  PROC DrawPart288()
    MoveL Offs(pOrigin,140.46,85.96,6.00),v60,z5,tPen\WObj:=wPaper;
    MoveL Offs(pOrigin,136.24,84.26,6.00),vTravel,z5,tPen\WObj:=wPaper;
    MoveL Offs(pOrigin,136.24,84.26,0.00),v60,z0,tPen\WObj:=wPaper;
    MoveL Offs(pOrigin,134.58,82.61,0.00),v40,z0,tPen\WObj:=wPaper;
    MoveL Offs(pOrigin,134.40,83.64,0.00),v40,z0,tPen\WObj:=wPaper;
    MoveL Offs(pOrigin,127.18,83.64,0.00),v40,z0,tPen\WObj:=wPaper;
    MoveL Offs(pOrigin,127.70,84.68,0.00),v40,z0,tPen\WObj:=wPaper;
    MoveL Offs(pOrigin,123.49,80.48,0.00),v40,fine,tPen\WObj:=wPaper;
    MoveL Offs(pOrigin,123.49,80.48,6.00),v60,z5,tPen\WObj:=wPaper;
    MoveL Offs(pOrigin,124.41,82.58,6.00),vTravel,z5,tPen\WObj:=wPaper;
    MoveL Offs(pOrigin,124.41,82.58,0.00),v60,z0,tPen\WObj:=wPaper;
    MoveL Offs(pOrigin,130.57,82.58,0.00),v40,z0,tPen\WObj:=wPaper;
    MoveL Offs(pOrigin,130.51,81.80,0.00),v40,z0,tPen\WObj:=wPaper;
    MoveL Offs(pOrigin,127.35,84.96,0.00),v40,fine,tPen\WObj:=wPaper;
    MoveL Offs(pOrigin,127.35,84.96,6.00),v60,z5,tPen\WObj:=wPaper;
    MoveL Offs(pOrigin,125.90,82.35,6.00),vTravel,z5,tPen\WObj:=wPaper;
    MoveL Offs(pOrigin,125.90,82.35,0.00),v60,z0,tPen\WObj:=wPaper;
    MoveL Offs(pOrigin,125.69,81.85,0.00),v40,z0,tPen\WObj:=wPaper;
    MoveL Offs(pOrigin,122.07,80.08,0.00),v40,z0,tPen\WObj:=wPaper;
    MoveL Offs(pOrigin,118.25,77.68,0.00),v40,z0,tPen\WObj:=wPaper;
    MoveL Offs(pOrigin,112.72,73.00,0.00),v40,fine,tPen\WObj:=wPaper;
    MoveL Offs(pOrigin,112.72,73.00,6.00),v60,z5,tPen\WObj:=wPaper;
    MoveL Offs(pOrigin,108.90,73.00,6.00),vTravel,z5,tPen\WObj:=wPaper;
    MoveL Offs(pOrigin,108.90,73.00,0.00),v60,z0,tPen\WObj:=wPaper;
    MoveL Offs(pOrigin,109.11,73.43,0.00),v40,z0,tPen\WObj:=wPaper;
    MoveL Offs(pOrigin,108.90,73.00,0.00),v40,fine,tPen\WObj:=wPaper;
    MoveL Offs(pOrigin,108.90,73.00,6.00),v60,z5,tPen\WObj:=wPaper;
    MoveL Offs(pOrigin,106.27,71.69,6.00),vTravel,z5,tPen\WObj:=wPaper;
    MoveL Offs(pOrigin,106.27,71.69,0.00),v60,z0,tPen\WObj:=wPaper;
    MoveL Offs(pOrigin,107.62,70.34,0.00),v40,z0,tPen\WObj:=wPaper;
    MoveL Offs(pOrigin,106.88,69.59,0.00),v40,z0,tPen\WObj:=wPaper;
    MoveL Offs(pOrigin,105.68,70.80,0.00),v40,z0,tPen\WObj:=wPaper;
    MoveL Offs(pOrigin,104.93,70.05,0.00),v40,z0,tPen\WObj:=wPaper;
    MoveL Offs(pOrigin,106.13,68.85,0.00),v40,z0,tPen\WObj:=wPaper;
    MoveL Offs(pOrigin,105.53,67.95,0.00),v40,z0,tPen\WObj:=wPaper;
    MoveL Offs(pOrigin,104.18,69.30,0.00),v40,fine,tPen\WObj:=wPaper;
    MoveL Offs(pOrigin,104.18,69.30,6.00),v60,z5,tPen\WObj:=wPaper;
    MoveL Offs(pOrigin,104.64,67.35,6.00),vTravel,z5,tPen\WObj:=wPaper;
    MoveL Offs(pOrigin,104.64,67.35,0.00),v60,z0,tPen\WObj:=wPaper;
    MoveL Offs(pOrigin,101.18,70.81,0.00),v40,z0,tPen\WObj:=wPaper;
    MoveL Offs(pOrigin,101.29,70.22,0.00),v40,z0,tPen\WObj:=wPaper;
    MoveL Offs(pOrigin,103.69,72.63,0.00),v40,fine,tPen\WObj:=wPaper;
    MoveL Offs(pOrigin,103.69,72.63,6.00),v60,z5,tPen\WObj:=wPaper;
    MoveL Offs(pOrigin,104.77,73.20,6.00),vTravel,z5,tPen\WObj:=wPaper;
    MoveL Offs(pOrigin,104.77,73.20,0.00),v60,z0,tPen\WObj:=wPaper;
    MoveL Offs(pOrigin,103.27,74.70,0.00),v40,z0,tPen\WObj:=wPaper;
    MoveL Offs(pOrigin,103.86,75.59,0.00),v40,z0,tPen\WObj:=wPaper;
    MoveL Offs(pOrigin,105.37,74.09,0.00),v40,z0,tPen\WObj:=wPaper;
    MoveL Offs(pOrigin,105.96,74.99,0.00),v40,z0,tPen\WObj:=wPaper;
    MoveL Offs(pOrigin,104.46,76.49,0.00),v40,fine,tPen\WObj:=wPaper;
    MoveL Offs(pOrigin,104.46,76.49,6.00),v60,z5,tPen\WObj:=wPaper;
    MoveL Offs(pOrigin,101.04,77.89,6.00),vTravel,z5,tPen\WObj:=wPaper;
    MoveL Offs(pOrigin,101.04,77.89,0.00),v60,z0,tPen\WObj:=wPaper;
    MoveL Offs(pOrigin,100.61,76.61,0.00),v40,z0,tPen\WObj:=wPaper;
    MoveL Offs(pOrigin,95.51,71.16,0.00),v40,z0,tPen\WObj:=wPaper;
    MoveL Offs(pOrigin,94.52,70.66,0.00),v40,z0,tPen\WObj:=wPaper;
    MoveL Offs(pOrigin,92.89,67.69,0.00),v40,z0,tPen\WObj:=wPaper;
    MoveL Offs(pOrigin,92.54,66.41,0.00),v40,z0,tPen\WObj:=wPaper;
    MoveL Offs(pOrigin,92.21,66.34,0.00),v40,z0,tPen\WObj:=wPaper;
    MoveL Offs(pOrigin,88.45,70.10,0.00),v40,fine,tPen\WObj:=wPaper;
    MoveL Offs(pOrigin,88.45,70.10,6.00),v60,z5,tPen\WObj:=wPaper;
    MoveL Offs(pOrigin,88.60,71.45,6.00),vTravel,z5,tPen\WObj:=wPaper;
    MoveL Offs(pOrigin,88.60,71.45,0.00),v60,z0,tPen\WObj:=wPaper;
    MoveL Offs(pOrigin,93.25,66.79,0.00),v40,fine,tPen\WObj:=wPaper;
    MoveL Offs(pOrigin,93.25,66.79,6.00),v60,z5,tPen\WObj:=wPaper;
    MoveL Offs(pOrigin,91.76,65.30,6.00),vTravel,z5,tPen\WObj:=wPaper;
    MoveL Offs(pOrigin,91.76,65.30,0.00),v60,z0,tPen\WObj:=wPaper;
    MoveL Offs(pOrigin,88.46,68.60,0.00),v40,z0,tPen\WObj:=wPaper;
    MoveL Offs(pOrigin,89.35,68.86,0.00),v40,z0,tPen\WObj:=wPaper;
    MoveL Offs(pOrigin,90.84,68.86,0.00),v40,fine,tPen\WObj:=wPaper;
    MoveL Offs(pOrigin,90.84,68.86,6.00),v60,z5,tPen\WObj:=wPaper;
    MoveL Offs(pOrigin,88.31,67.25,6.00),vTravel,z5,tPen\WObj:=wPaper;
    MoveL Offs(pOrigin,88.31,67.25,0.00),v60,z0,tPen\WObj:=wPaper;
    MoveL Offs(pOrigin,91.92,63.65,0.00),v40,fine,tPen\WObj:=wPaper;
    MoveL Offs(pOrigin,91.92,63.65,6.00),v60,z5,tPen\WObj:=wPaper;
    MoveL Offs(pOrigin,92.37,61.70,6.00),vTravel,z5,tPen\WObj:=wPaper;
    MoveL Offs(pOrigin,92.37,61.70,0.00),v60,z0,tPen\WObj:=wPaper;
    MoveL Offs(pOrigin,88.46,65.61,0.00),v40,z0,tPen\WObj:=wPaper;
    MoveL Offs(pOrigin,89.35,65.69,0.00),v40,z0,tPen\WObj:=wPaper;
    MoveL Offs(pOrigin,90.84,65.69,0.00),v40,fine,tPen\WObj:=wPaper;
    MoveL Offs(pOrigin,90.84,65.69,6.00),v60,z5,tPen\WObj:=wPaper;
    MoveL Offs(pOrigin,94.77,62.29,6.00),vTravel,z5,tPen\WObj:=wPaper;
    MoveL Offs(pOrigin,94.77,62.29,0.00),v60,z0,tPen\WObj:=wPaper;
    MoveL Offs(pOrigin,98.22,58.83,0.00),v40,z0,tPen\WObj:=wPaper;
    MoveL Offs(pOrigin,97.36,58.82,0.00),v40,z0,tPen\WObj:=wPaper;
    MoveL Offs(pOrigin,91.80,53.26,0.00),v40,z0,tPen\WObj:=wPaper;
    MoveL Offs(pOrigin,92.32,53.02,0.00),v40,z0,tPen\WObj:=wPaper;
    MoveL Offs(pOrigin,94.66,53.02,0.00),v40,z0,tPen\WObj:=wPaper;
    MoveL Offs(pOrigin,95.55,52.55,0.00),v40,z0,tPen\WObj:=wPaper;
    MoveL Offs(pOrigin,89.54,58.56,0.00),v40,fine,tPen\WObj:=wPaper;
    MoveL Offs(pOrigin,89.54,58.56,6.00),v60,z5,tPen\WObj:=wPaper;
    MoveL Offs(pOrigin,91.05,57.24,6.00),vTravel,z5,tPen\WObj:=wPaper;
    MoveL Offs(pOrigin,91.05,57.24,0.00),v60,z0,tPen\WObj:=wPaper;
    MoveL Offs(pOrigin,95.30,57.24,0.00),v40,z0,tPen\WObj:=wPaper;
    MoveL Offs(pOrigin,95.30,56.18,0.00),v40,z0,tPen\WObj:=wPaper;
    MoveL Offs(pOrigin,91.48,56.18,0.00),v40,z0,tPen\WObj:=wPaper;
    MoveL Offs(pOrigin,91.06,55.51,0.00),v40,z0,tPen\WObj:=wPaper;
    MoveL Offs(pOrigin,101.13,65.58,0.00),v40,z0,tPen\WObj:=wPaper;
    MoveL Offs(pOrigin,102.10,65.41,0.00),v40,z0,tPen\WObj:=wPaper;
    MoveL Offs(pOrigin,99.54,67.97,0.00),v40,z0,tPen\WObj:=wPaper;
    MoveL Offs(pOrigin,100.14,68.87,0.00),v40,z0,tPen\WObj:=wPaper;
    MoveL Offs(pOrigin,102.84,66.16,0.00),v40,z0,tPen\WObj:=wPaper;
    MoveL Offs(pOrigin,103.74,66.76,0.00),v40,z0,tPen\WObj:=wPaper;
    MoveL Offs(pOrigin,100.74,69.76,0.00),v40,fine,tPen\WObj:=wPaper;
    MoveL Offs(pOrigin,100.74,69.76,6.00),v60,z5,tPen\WObj:=wPaper;
    MoveL Offs(pOrigin,101.58,67.53,6.00),vTravel,z5,tPen\WObj:=wPaper;
    MoveL Offs(pOrigin,101.58,67.53,0.00),v60,z0,tPen\WObj:=wPaper;
    MoveL Offs(pOrigin,90.76,56.71,0.00),v40,z0,tPen\WObj:=wPaper;
    MoveL Offs(pOrigin,90.29,56.31,0.00),v40,z0,tPen\WObj:=wPaper;
    MoveL Offs(pOrigin,95.25,51.35,0.00),v40,fine,tPen\WObj:=wPaper;
    MoveL Offs(pOrigin,95.25,51.35,6.00),v60,z5,tPen\WObj:=wPaper;
    MoveL Offs(pOrigin,94.24,49.85,6.00),vTravel,z5,tPen\WObj:=wPaper;
    MoveL Offs(pOrigin,94.24,49.85,0.00),v60,z0,tPen\WObj:=wPaper;
    MoveL Offs(pOrigin,92.32,49.85,0.00),v40,fine,tPen\WObj:=wPaper;
    MoveL Offs(pOrigin,92.32,49.85,6.00),v60,z5,tPen\WObj:=wPaper;
    MoveL Offs(pOrigin,91.36,50.77,6.00),vTravel,z5,tPen\WObj:=wPaper;
    MoveL Offs(pOrigin,91.36,50.77,0.00),v60,z0,tPen\WObj:=wPaper;
    MoveL Offs(pOrigin,95.56,46.56,0.00),v40,z0,tPen\WObj:=wPaper;
    MoveL Offs(pOrigin,94.45,46.68,0.00),v40,z0,tPen\WObj:=wPaper;
    MoveL Offs(pOrigin,93.18,46.68,0.00),v40,fine,tPen\WObj:=wPaper;
  ENDPROC

  PROC DrawPart289()
    MoveL Offs(pOrigin,93.18,46.68,6.00),v60,z5,tPen\WObj:=wPaper;
    MoveL Offs(pOrigin,94.24,44.57,6.00),vTravel,z5,tPen\WObj:=wPaper;
    MoveL Offs(pOrigin,94.24,44.57,0.00),v60,z0,tPen\WObj:=wPaper;
    MoveL Offs(pOrigin,95.94,44.57,0.00),v40,z0,tPen\WObj:=wPaper;
    MoveL Offs(pOrigin,96.57,44.59,0.00),v40,z0,tPen\WObj:=wPaper;
    MoveL Offs(pOrigin,95.22,43.24,0.00),v40,z0,tPen\WObj:=wPaper;
    MoveL Offs(pOrigin,95.30,43.51,0.00),v40,z0,tPen\WObj:=wPaper;
    MoveL Offs(pOrigin,97.00,43.51,0.00),v40,z0,tPen\WObj:=wPaper;
    MoveL Offs(pOrigin,97.00,43.67,0.00),v40,z0,tPen\WObj:=wPaper;
    MoveL Offs(pOrigin,95.51,45.16,0.00),v40,z0,tPen\WObj:=wPaper;
    MoveL Offs(pOrigin,97.00,43.67,0.00),v40,z0,tPen\WObj:=wPaper;
    MoveL Offs(pOrigin,97.46,43.99,0.00),v40,z0,tPen\WObj:=wPaper;
    MoveL Offs(pOrigin,95.81,42.34,0.00),v40,z0,tPen\WObj:=wPaper;
    MoveL Offs(pOrigin,95.94,42.61,0.00),v40,z0,tPen\WObj:=wPaper;
    MoveL Offs(pOrigin,94.03,44.53,0.00),v40,z0,tPen\WObj:=wPaper;
    MoveL Offs(pOrigin,95.94,42.61,0.00),v40,fine,tPen\WObj:=wPaper;
    MoveL Offs(pOrigin,95.94,42.61,6.00),v60,z5,tPen\WObj:=wPaper;
    MoveL Offs(pOrigin,97.64,41.55,6.00),vTravel,z5,tPen\WObj:=wPaper;
    MoveL Offs(pOrigin,97.64,41.55,0.00),v60,z0,tPen\WObj:=wPaper;
    MoveL Offs(pOrigin,99.55,40.42,0.00),v40,z0,tPen\WObj:=wPaper;
    MoveL Offs(pOrigin,106.35,38.58,0.00),v40,z0,tPen\WObj:=wPaper;
    MoveL Offs(pOrigin,106.67,39.00,0.00),v40,z0,tPen\WObj:=wPaper;
    MoveL Offs(pOrigin,106.67,40.06,0.00),v40,fine,tPen\WObj:=wPaper;
    MoveL Offs(pOrigin,106.67,40.06,6.00),v60,z5,tPen\WObj:=wPaper;
    MoveL Offs(pOrigin,108.78,40.49,6.00),vTravel,z5,tPen\WObj:=wPaper;
    MoveL Offs(pOrigin,108.78,40.49,0.00),v60,z0,tPen\WObj:=wPaper;
    MoveL Offs(pOrigin,108.78,37.72,0.00),v40,z0,tPen\WObj:=wPaper;
    MoveL Offs(pOrigin,109.84,37.72,0.00),v40,z0,tPen\WObj:=wPaper;
    MoveL Offs(pOrigin,109.84,39.85,0.00),v40,fine,tPen\WObj:=wPaper;
    MoveL Offs(pOrigin,109.84,39.85,6.00),v60,z5,tPen\WObj:=wPaper;
    MoveL Offs(pOrigin,109.44,41.04,6.00),vTravel,z5,tPen\WObj:=wPaper;
    MoveL Offs(pOrigin,109.44,41.04,0.00),v60,z0,tPen\WObj:=wPaper;
    MoveL Offs(pOrigin,104.48,36.08,0.00),v40,fine,tPen\WObj:=wPaper;
    MoveL Offs(pOrigin,104.48,36.08,6.00),v60,z5,tPen\WObj:=wPaper;
    MoveL Offs(pOrigin,103.69,33.95,6.00),vTravel,z5,tPen\WObj:=wPaper;
    MoveL Offs(pOrigin,103.69,33.95,0.00),v60,z0,tPen\WObj:=wPaper;
    MoveL Offs(pOrigin,100.24,37.41,0.00),v40,fine,tPen\WObj:=wPaper;
    MoveL Offs(pOrigin,100.24,37.41,6.00),v60,z5,tPen\WObj:=wPaper;
    MoveL Offs(pOrigin,100.75,39.81,6.00),vTravel,z5,tPen\WObj:=wPaper;
    MoveL Offs(pOrigin,100.75,39.81,0.00),v60,z0,tPen\WObj:=wPaper;
    MoveL Offs(pOrigin,102.25,41.31,0.00),v40,fine,tPen\WObj:=wPaper;
    MoveL Offs(pOrigin,102.25,41.31,6.00),v60,z5,tPen\WObj:=wPaper;
    MoveL Offs(pOrigin,103.45,41.02,6.00),vTravel,z5,tPen\WObj:=wPaper;
    MoveL Offs(pOrigin,103.45,41.02,0.00),v60,z0,tPen\WObj:=wPaper;
    MoveL Offs(pOrigin,101.94,39.51,0.00),v40,fine,tPen\WObj:=wPaper;
    MoveL Offs(pOrigin,101.94,39.51,6.00),v60,z5,tPen\WObj:=wPaper;
    MoveL Offs(pOrigin,103.82,41.29,6.00),vTravel,z5,tPen\WObj:=wPaper;
    MoveL Offs(pOrigin,103.82,41.29,0.00),v60,z0,tPen\WObj:=wPaper;
    MoveL Offs(pOrigin,110.58,34.53,0.00),v40,fine,tPen\WObj:=wPaper;
    MoveL Offs(pOrigin,110.58,34.53,6.00),v60,z5,tPen\WObj:=wPaper;
    MoveL Offs(pOrigin,113.17,37.30,6.00),vTravel,z5,tPen\WObj:=wPaper;
    MoveL Offs(pOrigin,113.17,37.30,0.00),v60,z0,tPen\WObj:=wPaper;
    MoveL Offs(pOrigin,117.83,41.96,0.00),v40,fine,tPen\WObj:=wPaper;
    MoveL Offs(pOrigin,117.83,41.96,6.00),v60,z5,tPen\WObj:=wPaper;
    MoveL Offs(pOrigin,118.13,40.76,6.00),vTravel,z5,tPen\WObj:=wPaper;
    MoveL Offs(pOrigin,118.13,40.76,0.00),v60,z0,tPen\WObj:=wPaper;
    MoveL Offs(pOrigin,114.97,37.61,0.00),v40,z0,tPen\WObj:=wPaper;
    MoveL Offs(pOrigin,115.12,38.57,0.00),v40,z0,tPen\WObj:=wPaper;
    MoveL Offs(pOrigin,115.12,39.64,0.00),v40,z0,tPen\WObj:=wPaper;
    MoveL Offs(pOrigin,114.06,39.64,0.00),v40,z0,tPen\WObj:=wPaper;
    MoveL Offs(pOrigin,114.06,38.36,0.00),v40,fine,tPen\WObj:=wPaper;
    MoveL Offs(pOrigin,114.06,38.36,6.00),v60,z5,tPen\WObj:=wPaper;
    MoveL Offs(pOrigin,115.06,40.91,6.00),vTravel,z5,tPen\WObj:=wPaper;
    MoveL Offs(pOrigin,115.06,40.91,0.00),v60,z0,tPen\WObj:=wPaper;
    MoveL Offs(pOrigin,116.55,39.42,0.00),v40,z0,tPen\WObj:=wPaper;
    MoveL Offs(pOrigin,117.12,39.64,0.00),v40,z0,tPen\WObj:=wPaper;
    MoveL Offs(pOrigin,117.19,40.49,0.00),v40,fine,tPen\WObj:=wPaper;
    MoveL Offs(pOrigin,117.19,40.49,6.00),v60,z5,tPen\WObj:=wPaper;
    MoveL Offs(pOrigin,115.06,40.91,6.00),vTravel,z5,tPen\WObj:=wPaper;
    MoveL Offs(pOrigin,115.06,40.91,0.00),v60,z0,tPen\WObj:=wPaper;
    MoveL Offs(pOrigin,114.50,40.70,0.00),v40,z0,tPen\WObj:=wPaper;
    MoveL Offs(pOrigin,114.21,39.92,0.00),v40,z0,tPen\WObj:=wPaper;
    MoveL Offs(pOrigin,113.57,40.13,0.00),v40,z0,tPen\WObj:=wPaper;
    MoveL Offs(pOrigin,112.30,41.76,0.00),v40,fine,tPen\WObj:=wPaper;
    MoveL Offs(pOrigin,112.30,41.76,6.00),v60,z5,tPen\WObj:=wPaper;
    MoveL Offs(pOrigin,112.30,43.89,6.00),vTravel,z5,tPen\WObj:=wPaper;
    MoveL Offs(pOrigin,112.30,43.89,0.00),v60,z0,tPen\WObj:=wPaper;
    MoveL Offs(pOrigin,113.57,44.31,0.00),v40,fine,tPen\WObj:=wPaper;
    MoveL Offs(pOrigin,113.57,44.31,6.00),v60,z5,tPen\WObj:=wPaper;
    MoveL Offs(pOrigin,114.44,45.60,6.00),vTravel,z5,tPen\WObj:=wPaper;
    MoveL Offs(pOrigin,114.44,45.60,0.00),v60,z0,tPen\WObj:=wPaper;
    MoveL Offs(pOrigin,124.06,35.99,0.00),v40,fine,tPen\WObj:=wPaper;
    MoveL Offs(pOrigin,124.06,35.99,6.00),v60,z5,tPen\WObj:=wPaper;
    MoveL Offs(pOrigin,123.51,37.18,6.00),vTravel,z5,tPen\WObj:=wPaper;
    MoveL Offs(pOrigin,123.51,37.18,0.00),v60,z0,tPen\WObj:=wPaper;
    MoveL Offs(pOrigin,129.07,42.74,0.00),v40,z0,tPen\WObj:=wPaper;
    MoveL Offs(pOrigin,129.81,42.00,0.00),v40,z0,tPen\WObj:=wPaper;
    MoveL Offs(pOrigin,125.01,37.19,0.00),v40,z0,tPen\WObj:=wPaper;
    MoveL Offs(pOrigin,125.41,36.13,0.00),v40,z0,tPen\WObj:=wPaper;
    MoveL Offs(pOrigin,119.10,42.44,0.00),v40,z0,tPen\WObj:=wPaper;
    MoveL Offs(pOrigin,119.78,42.42,0.00),v40,z0,tPen\WObj:=wPaper;
    MoveL Offs(pOrigin,122.03,44.67,0.00),v40,z0,tPen\WObj:=wPaper;
    MoveL Offs(pOrigin,121.65,44.57,0.00),v40,z0,tPen\WObj:=wPaper;
    MoveL Offs(pOrigin,119.74,44.57,0.00),v40,z0,tPen\WObj:=wPaper;
    MoveL Offs(pOrigin,118.79,44.24,0.00),v40,z0,tPen\WObj:=wPaper;
    MoveL Offs(pOrigin,126.75,36.28,0.00),v40,z0,tPen\WObj:=wPaper;
    MoveL Offs(pOrigin,126.50,37.19,0.00),v40,z0,tPen\WObj:=wPaper;
    MoveL Offs(pOrigin,130.71,41.40,0.00),v40,z0,tPen\WObj:=wPaper;
    MoveL Offs(pOrigin,130.36,41.12,0.00),v40,z0,tPen\WObj:=wPaper;
    MoveL Offs(pOrigin,129.94,41.55,0.00),v40,z0,tPen\WObj:=wPaper;
    MoveL Offs(pOrigin,130.36,41.12,0.00),v40,z0,tPen\WObj:=wPaper;
    MoveL Offs(pOrigin,129.90,40.91,0.00),v40,z0,tPen\WObj:=wPaper;
    MoveL Offs(pOrigin,129.90,38.15,0.00),v40,z0,tPen\WObj:=wPaper;
    MoveL Offs(pOrigin,130.96,37.72,0.00),v40,z0,tPen\WObj:=wPaper;
    MoveL Offs(pOrigin,130.96,40.28,0.00),v40,z0,tPen\WObj:=wPaper;
    MoveL Offs(pOrigin,131.64,40.34,0.00),v40,z0,tPen\WObj:=wPaper;
    MoveL Offs(pOrigin,120.38,40.34,0.00),v40,z0,tPen\WObj:=wPaper;
    MoveL Offs(pOrigin,120.38,41.40,0.00),v40,z0,tPen\WObj:=wPaper;
    MoveL Offs(pOrigin,123.56,41.40,0.00),v40,z0,tPen\WObj:=wPaper;
    MoveL Offs(pOrigin,123.67,41.83,0.00),v40,z0,tPen\WObj:=wPaper;
    MoveL Offs(pOrigin,119.92,38.07,0.00),v40,z0,tPen\WObj:=wPaper;
    MoveL Offs(pOrigin,118.89,38.23,0.00),v40,z0,tPen\WObj:=wPaper;
    MoveL Offs(pOrigin,105.29,38.23,0.00),v40,fine,tPen\WObj:=wPaper;
    MoveL Offs(pOrigin,105.29,38.23,6.00),v60,z5,tPen\WObj:=wPaper;
    MoveL Offs(pOrigin,104.81,45.37,6.00),vTravel,z5,tPen\WObj:=wPaper;
    MoveL Offs(pOrigin,104.81,45.37,0.00),v60,z0,tPen\WObj:=wPaper;
    MoveL Offs(pOrigin,106.01,46.57,0.00),v40,fine,tPen\WObj:=wPaper;
    MoveL Offs(pOrigin,106.01,46.57,6.00),v60,z5,tPen\WObj:=wPaper;
    MoveL Offs(pOrigin,104.11,45.48,6.00),vTravel,z5,tPen\WObj:=wPaper;
    MoveL Offs(pOrigin,104.11,45.48,0.00),v60,z0,tPen\WObj:=wPaper;
  ENDPROC

  PROC DrawPart290()
    MoveL Offs(pOrigin,114.62,34.97,0.00),v40,fine,tPen\WObj:=wPaper;
    MoveL Offs(pOrigin,114.62,34.97,6.00),v60,z5,tPen\WObj:=wPaper;
    MoveL Offs(pOrigin,118.12,37.77,6.00),vTravel,z5,tPen\WObj:=wPaper;
    MoveL Offs(pOrigin,118.12,37.77,0.00),v60,z0,tPen\WObj:=wPaper;
    MoveL Offs(pOrigin,123.08,42.73,0.00),v40,z0,tPen\WObj:=wPaper;
    MoveL Offs(pOrigin,123.14,42.19,0.00),v40,z0,tPen\WObj:=wPaper;
    MoveL Offs(pOrigin,122.71,42.61,0.00),v40,z0,tPen\WObj:=wPaper;
    MoveL Offs(pOrigin,123.14,42.19,0.00),v40,z0,tPen\WObj:=wPaper;
    MoveL Offs(pOrigin,122.50,43.04,0.00),v40,z0,tPen\WObj:=wPaper;
    MoveL Offs(pOrigin,122.29,43.46,0.00),v40,z0,tPen\WObj:=wPaper;
    MoveL Offs(pOrigin,122.50,43.04,0.00),v40,z0,tPen\WObj:=wPaper;
    MoveL Offs(pOrigin,122.07,43.89,0.00),v40,z0,tPen\WObj:=wPaper;
    MoveL Offs(pOrigin,121.86,44.31,0.00),v40,z0,tPen\WObj:=wPaper;
    MoveL Offs(pOrigin,122.07,43.89,0.00),v40,z0,tPen\WObj:=wPaper;
    MoveL Offs(pOrigin,121.45,43.89,0.00),v40,z0,tPen\WObj:=wPaper;
    MoveL Offs(pOrigin,121.45,39.21,0.00),v40,z0,tPen\WObj:=wPaper;
    MoveL Offs(pOrigin,121.56,38.23,0.00),v40,z0,tPen\WObj:=wPaper;
    MoveL Offs(pOrigin,127.42,44.09,0.00),v40,fine,tPen\WObj:=wPaper;
    MoveL Offs(pOrigin,127.42,44.09,6.00),v60,z5,tPen\WObj:=wPaper;
    MoveL Offs(pOrigin,128.85,41.55,6.00),vTravel,z5,tPen\WObj:=wPaper;
    MoveL Offs(pOrigin,128.85,41.55,0.00),v60,z0,tPen\WObj:=wPaper;
    MoveL Offs(pOrigin,128.85,39.00,0.00),v40,z0,tPen\WObj:=wPaper;
    MoveL Offs(pOrigin,128.66,38.23,0.00),v40,z0,tPen\WObj:=wPaper;
    MoveL Offs(pOrigin,136.31,38.23,0.00),v40,z0,tPen\WObj:=wPaper;
    MoveL Offs(pOrigin,136.84,38.57,0.00),v40,z0,tPen\WObj:=wPaper;
    MoveL Offs(pOrigin,134.89,36.62,0.00),v40,z0,tPen\WObj:=wPaper;
    MoveL Offs(pOrigin,134.39,36.10,0.00),v40,z0,tPen\WObj:=wPaper;
    MoveL Offs(pOrigin,123.12,47.37,0.00),v40,fine,tPen\WObj:=wPaper;
    MoveL Offs(pOrigin,123.12,47.37,6.00),v60,z5,tPen\WObj:=wPaper;
    MoveL Offs(pOrigin,123.28,45.72,6.00),vTravel,z5,tPen\WObj:=wPaper;
    MoveL Offs(pOrigin,123.28,45.72,0.00),v60,z0,tPen\WObj:=wPaper;
    MoveL Offs(pOrigin,132.90,36.11,0.00),v40,z0,tPen\WObj:=wPaper;
    MoveL Offs(pOrigin,132.20,36.91,0.00),v40,z0,tPen\WObj:=wPaper;
    MoveL Offs(pOrigin,134.60,39.32,0.00),v40,z0,tPen\WObj:=wPaper;
    MoveL Offs(pOrigin,133.55,39.76,0.00),v40,z0,tPen\WObj:=wPaper;
    MoveL Offs(pOrigin,131.00,37.21,0.00),v40,z0,tPen\WObj:=wPaper;
    MoveL Offs(pOrigin,132.01,37.51,0.00),v40,z0,tPen\WObj:=wPaper;
    MoveL Offs(pOrigin,132.01,39.85,0.00),v40,z0,tPen\WObj:=wPaper;
    MoveL Offs(pOrigin,132.70,40.06,0.00),v40,z0,tPen\WObj:=wPaper;
    MoveL Offs(pOrigin,135.04,38.93,0.00),v40,z0,tPen\WObj:=wPaper;
    MoveL Offs(pOrigin,139.50,37.72,0.00),v40,z0,tPen\WObj:=wPaper;
    MoveL Offs(pOrigin,141.20,37.51,0.00),v40,z0,tPen\WObj:=wPaper;
    MoveL Offs(pOrigin,141.84,38.36,0.00),v40,fine,tPen\WObj:=wPaper;
    MoveL Offs(pOrigin,141.84,38.36,6.00),v60,z5,tPen\WObj:=wPaper;
    MoveL Offs(pOrigin,142.69,39.94,6.00),vTravel,z5,tPen\WObj:=wPaper;
    MoveL Offs(pOrigin,142.69,39.94,0.00),v60,z0,tPen\WObj:=wPaper;
    MoveL Offs(pOrigin,145.85,43.09,0.00),v40,z0,tPen\WObj:=wPaper;
    MoveL Offs(pOrigin,146.09,42.61,0.00),v40,z0,tPen\WObj:=wPaper;
    MoveL Offs(pOrigin,144.60,44.10,0.00),v40,z0,tPen\WObj:=wPaper;
    MoveL Offs(pOrigin,146.09,42.61,0.00),v40,fine,tPen\WObj:=wPaper;
    MoveL Offs(pOrigin,146.09,42.61,6.00),v60,z5,tPen\WObj:=wPaper;
    MoveL Offs(pOrigin,146.05,43.86,6.00),vTravel,z5,tPen\WObj:=wPaper;
    MoveL Offs(pOrigin,146.05,43.86,0.00),v60,z0,tPen\WObj:=wPaper;
    MoveL Offs(pOrigin,135.09,54.83,0.00),v40,fine,tPen\WObj:=wPaper;
    MoveL Offs(pOrigin,135.09,54.83,6.00),v60,z5,tPen\WObj:=wPaper;
    MoveL Offs(pOrigin,134.94,51.98,6.00),vTravel,z5,tPen\WObj:=wPaper;
    MoveL Offs(pOrigin,134.94,51.98,0.00),v60,z0,tPen\WObj:=wPaper;
    MoveL Offs(pOrigin,151.62,35.30,0.00),v40,fine,tPen\WObj:=wPaper;
    MoveL Offs(pOrigin,151.62,35.30,6.00),v60,z5,tPen\WObj:=wPaper;
    MoveL Offs(pOrigin,150.43,35.01,6.00),vTravel,z5,tPen\WObj:=wPaper;
    MoveL Offs(pOrigin,150.43,35.01,0.00),v60,z0,tPen\WObj:=wPaper;
    MoveL Offs(pOrigin,135.10,50.33,0.00),v40,fine,tPen\WObj:=wPaper;
    MoveL Offs(pOrigin,135.10,50.33,6.00),v60,z5,tPen\WObj:=wPaper;
    MoveL Offs(pOrigin,136.43,48.61,6.00),vTravel,z5,tPen\WObj:=wPaper;
    MoveL Offs(pOrigin,136.43,48.61,0.00),v60,z0,tPen\WObj:=wPaper;
    MoveL Offs(pOrigin,148.15,60.33,0.00),v40,z0,tPen\WObj:=wPaper;
    MoveL Offs(pOrigin,147.57,60.41,0.00),v40,z0,tPen\WObj:=wPaper;
    MoveL Offs(pOrigin,138.86,60.41,0.00),v40,z0,tPen\WObj:=wPaper;
    MoveL Offs(pOrigin,138.11,60.75,0.00),v40,z0,tPen\WObj:=wPaper;
    MoveL Offs(pOrigin,143.67,66.31,0.00),v40,z0,tPen\WObj:=wPaper;
    MoveL Offs(pOrigin,143.14,66.19,0.00),v40,z0,tPen\WObj:=wPaper;
    MoveL Offs(pOrigin,149.15,60.18,0.00),v40,z0,tPen\WObj:=wPaper;
    MoveL Offs(pOrigin,149.90,60.92,0.00),v40,z0,tPen\WObj:=wPaper;
    MoveL Offs(pOrigin,143.89,66.93,0.00),v40,z0,tPen\WObj:=wPaper;
    MoveL Offs(pOrigin,144.78,67.53,0.00),v40,z0,tPen\WObj:=wPaper;
    MoveL Offs(pOrigin,150.49,61.82,0.00),v40,z0,tPen\WObj:=wPaper;
    MoveL Offs(pOrigin,150.12,62.38,0.00),v40,z0,tPen\WObj:=wPaper;
    MoveL Offs(pOrigin,150.98,63.22,0.00),v40,z0,tPen\WObj:=wPaper;
    MoveL Offs(pOrigin,150.12,62.38,0.00),v40,z0,tPen\WObj:=wPaper;
    MoveL Offs(pOrigin,149.49,62.52,0.00),v40,z0,tPen\WObj:=wPaper;
    MoveL Offs(pOrigin,140.56,62.52,0.00),v40,fine,tPen\WObj:=wPaper;
    MoveL Offs(pOrigin,140.56,62.52,6.00),v60,z5,tPen\WObj:=wPaper;
    MoveL Offs(pOrigin,139.85,63.50,6.00),vTravel,z5,tPen\WObj:=wPaper;
    MoveL Offs(pOrigin,139.85,63.50,0.00),v60,z0,tPen\WObj:=wPaper;
    MoveL Offs(pOrigin,146.61,56.74,0.00),v40,z0,tPen\WObj:=wPaper;
    MoveL Offs(pOrigin,147.21,57.64,0.00),v40,z0,tPen\WObj:=wPaper;
    MoveL Offs(pOrigin,140.75,64.10,0.00),v40,z0,tPen\WObj:=wPaper;
    MoveL Offs(pOrigin,141.62,63.58,0.00),v40,z0,tPen\WObj:=wPaper;
    MoveL Offs(pOrigin,150.34,63.58,0.00),v40,fine,tPen\WObj:=wPaper;
    MoveL Offs(pOrigin,150.34,63.58,6.00),v60,z5,tPen\WObj:=wPaper;
    MoveL Offs(pOrigin,151.24,62.57,6.00),vTravel,z5,tPen\WObj:=wPaper;
    MoveL Offs(pOrigin,151.24,62.57,0.00),v60,z0,tPen\WObj:=wPaper;
    MoveL Offs(pOrigin,145.68,68.13,0.00),v40,z0,tPen\WObj:=wPaper;
    MoveL Offs(pOrigin,146.58,68.72,0.00),v40,z0,tPen\WObj:=wPaper;
    MoveL Offs(pOrigin,151.99,63.31,0.00),v40,z0,tPen\WObj:=wPaper;
    MoveL Offs(pOrigin,152.58,64.21,0.00),v40,z0,tPen\WObj:=wPaper;
    MoveL Offs(pOrigin,147.47,69.32,0.00),v40,fine,tPen\WObj:=wPaper;
    MoveL Offs(pOrigin,147.47,69.32,6.00),v60,z5,tPen\WObj:=wPaper;
    MoveL Offs(pOrigin,147.85,68.11,6.00),vTravel,z5,tPen\WObj:=wPaper;
    MoveL Offs(pOrigin,147.85,68.11,0.00),v60,z0,tPen\WObj:=wPaper;
    MoveL Offs(pOrigin,147.85,65.99,0.00),v40,fine,tPen\WObj:=wPaper;
    MoveL Offs(pOrigin,147.85,65.99,6.00),v60,z5,tPen\WObj:=wPaper;
    MoveL Offs(pOrigin,148.00,64.50,6.00),vTravel,z5,tPen\WObj:=wPaper;
    MoveL Offs(pOrigin,148.00,64.50,0.00),v60,z0,tPen\WObj:=wPaper;
    MoveL Offs(pOrigin,149.06,65.56,0.00),v40,z0,tPen\WObj:=wPaper;
    MoveL Offs(pOrigin,148.00,64.50,0.00),v40,z0,tPen\WObj:=wPaper;
    MoveL Offs(pOrigin,148.91,64.07,0.00),v40,z0,tPen\WObj:=wPaper;
    MoveL Offs(pOrigin,148.91,63.01,0.00),v40,z0,tPen\WObj:=wPaper;
    MoveL Offs(pOrigin,147.85,63.01,0.00),v40,z0,tPen\WObj:=wPaper;
    MoveL Offs(pOrigin,147.85,61.74,0.00),v40,z0,tPen\WObj:=wPaper;
    MoveL Offs(pOrigin,148.43,61.46,0.00),v40,z0,tPen\WObj:=wPaper;
    MoveL Offs(pOrigin,139.71,61.46,0.00),v40,z0,tPen\WObj:=wPaper;
    MoveL Offs(pOrigin,139.36,61.67,0.00),v40,z0,tPen\WObj:=wPaper;
    MoveL Offs(pOrigin,142.26,64.50,0.00),v40,z0,tPen\WObj:=wPaper;
    MoveL Offs(pOrigin,139.36,61.67,0.00),v40,z0,tPen\WObj:=wPaper;
    MoveL Offs(pOrigin,138.51,61.86,0.00),v40,z0,tPen\WObj:=wPaper;
    MoveL Offs(pOrigin,145.57,54.79,0.00),v40,z0,tPen\WObj:=wPaper;
    MoveL Offs(pOrigin,146.17,55.69,0.00),v40,z0,tPen\WObj:=wPaper;
    MoveL Offs(pOrigin,139.26,62.60,0.00),v40,fine,tPen\WObj:=wPaper;
    MoveL Offs(pOrigin,139.26,62.60,6.00),v60,z5,tPen\WObj:=wPaper;
  ENDPROC

  PROC DrawPart291()
    MoveL Offs(pOrigin,137.91,60.96,6.00),vTravel,z5,tPen\WObj:=wPaper;
    MoveL Offs(pOrigin,137.91,60.96,0.00),v60,z0,tPen\WObj:=wPaper;
    MoveL Offs(pOrigin,145.13,53.75,0.00),v40,z0,tPen\WObj:=wPaper;
    MoveL Offs(pOrigin,144.18,54.07,0.00),v40,z0,tPen\WObj:=wPaper;
    MoveL Offs(pOrigin,138.44,54.07,0.00),v40,z0,tPen\WObj:=wPaper;
    MoveL Offs(pOrigin,138.35,53.24,0.00),v40,z0,tPen\WObj:=wPaper;
    MoveL Offs(pOrigin,138.35,50.69,0.00),v40,z0,tPen\WObj:=wPaper;
    MoveL Offs(pOrigin,139.41,50.48,0.00),v40,z0,tPen\WObj:=wPaper;
    MoveL Offs(pOrigin,139.41,54.94,0.00),v40,fine,tPen\WObj:=wPaper;
    MoveL Offs(pOrigin,139.41,54.94,6.00),v60,z5,tPen\WObj:=wPaper;
    MoveL Offs(pOrigin,140.56,54.30,6.00),vTravel,z5,tPen\WObj:=wPaper;
    MoveL Offs(pOrigin,140.56,54.30,0.00),v60,z0,tPen\WObj:=wPaper;
    MoveL Offs(pOrigin,142.40,58.76,0.00),v40,z0,tPen\WObj:=wPaper;
    MoveL Offs(pOrigin,143.75,60.67,0.00),v40,z0,tPen\WObj:=wPaper;
    MoveL Offs(pOrigin,145.02,61.31,0.00),v40,z0,tPen\WObj:=wPaper;
    MoveL Offs(pOrigin,148.85,65.56,0.00),v40,z0,tPen\WObj:=wPaper;
    MoveL Offs(pOrigin,152.25,67.90,0.00),v40,z0,tPen\WObj:=wPaper;
    MoveL Offs(pOrigin,152.08,67.90,0.00),v40,z0,tPen\WObj:=wPaper;
    MoveL Offs(pOrigin,152.08,70.24,0.00),v40,z0,tPen\WObj:=wPaper;
    MoveL Offs(pOrigin,151.02,69.81,0.00),v40,z0,tPen\WObj:=wPaper;
    MoveL Offs(pOrigin,151.02,67.47,0.00),v40,fine,tPen\WObj:=wPaper;
    MoveL Offs(pOrigin,151.02,67.47,6.00),v60,z5,tPen\WObj:=wPaper;
    MoveL Offs(pOrigin,152.89,68.54,6.00),vTravel,z5,tPen\WObj:=wPaper;
    MoveL Offs(pOrigin,152.89,68.54,0.00),v60,z0,tPen\WObj:=wPaper;
    MoveL Offs(pOrigin,153.10,68.96,0.00),v40,z0,tPen\WObj:=wPaper;
    MoveL Offs(pOrigin,152.89,68.54,0.00),v40,fine,tPen\WObj:=wPaper;
    MoveL Offs(pOrigin,152.89,68.54,6.00),v60,z5,tPen\WObj:=wPaper;
    MoveL Offs(pOrigin,153.13,66.62,6.00),vTravel,z5,tPen\WObj:=wPaper;
    MoveL Offs(pOrigin,153.13,66.62,0.00),v60,z0,tPen\WObj:=wPaper;
    MoveL Offs(pOrigin,153.13,70.66,0.00),v40,z0,tPen\WObj:=wPaper;
    MoveL Offs(pOrigin,154.19,70.88,0.00),v40,z0,tPen\WObj:=wPaper;
    MoveL Offs(pOrigin,154.19,67.05,0.00),v40,z0,tPen\WObj:=wPaper;
    MoveL Offs(pOrigin,154.38,66.41,0.00),v40,z0,tPen\WObj:=wPaper;
    MoveL Offs(pOrigin,154.80,66.62,0.00),v40,z0,tPen\WObj:=wPaper;
    MoveL Offs(pOrigin,154.38,66.41,0.00),v40,z0,tPen\WObj:=wPaper;
    MoveL Offs(pOrigin,153.52,65.99,0.00),v40,z0,tPen\WObj:=wPaper;
    MoveL Offs(pOrigin,153.95,66.20,0.00),v40,z0,tPen\WObj:=wPaper;
    MoveL Offs(pOrigin,153.52,65.99,0.00),v40,z0,tPen\WObj:=wPaper;
    MoveL Offs(pOrigin,153.10,65.69,0.00),v40,z0,tPen\WObj:=wPaper;
    MoveL Offs(pOrigin,143.96,65.69,0.00),v40,z0,tPen\WObj:=wPaper;
    MoveL Offs(pOrigin,143.63,65.14,0.00),v40,z0,tPen\WObj:=wPaper;
    MoveL Offs(pOrigin,143.63,61.52,0.00),v40,fine,tPen\WObj:=wPaper;
    MoveL Offs(pOrigin,143.63,61.52,6.00),v60,z5,tPen\WObj:=wPaper;
    MoveL Offs(pOrigin,142.57,60.46,6.00),vTravel,z5,tPen\WObj:=wPaper;
    MoveL Offs(pOrigin,142.57,60.46,0.00),v60,z0,tPen\WObj:=wPaper;
    MoveL Offs(pOrigin,142.57,64.07,0.00),v40,z0,tPen\WObj:=wPaper;
    MoveL Offs(pOrigin,142.90,64.63,0.00),v40,z0,tPen\WObj:=wPaper;
    MoveL Offs(pOrigin,151.61,64.63,0.00),v40,z0,tPen\WObj:=wPaper;
    MoveL Offs(pOrigin,152.25,65.14,0.00),v40,z0,tPen\WObj:=wPaper;
    MoveL Offs(pOrigin,152.89,65.56,0.00),v40,z0,tPen\WObj:=wPaper;
    MoveL Offs(pOrigin,152.25,65.14,0.00),v40,fine,tPen\WObj:=wPaper;
    MoveL Offs(pOrigin,152.25,65.14,6.00),v60,z5,tPen\WObj:=wPaper;
    MoveL Offs(pOrigin,154.53,65.25,6.00),vTravel,z5,tPen\WObj:=wPaper;
    MoveL Offs(pOrigin,154.53,65.25,0.00),v60,z0,tPen\WObj:=wPaper;
    MoveL Offs(pOrigin,149.42,70.36,0.00),v40,z0,tPen\WObj:=wPaper;
    MoveL Offs(pOrigin,150.47,70.81,0.00),v40,z0,tPen\WObj:=wPaper;
    MoveL Offs(pOrigin,155.42,65.85,0.00),v40,fine,tPen\WObj:=wPaper;
    MoveL Offs(pOrigin,155.42,65.85,6.00),v60,z5,tPen\WObj:=wPaper;
    MoveL Offs(pOrigin,157.52,66.74,6.00),vTravel,z5,tPen\WObj:=wPaper;
    MoveL Offs(pOrigin,157.52,66.74,0.00),v60,z0,tPen\WObj:=wPaper;
    MoveL Offs(pOrigin,152.41,71.85,0.00),v40,fine,tPen\WObj:=wPaper;
    MoveL Offs(pOrigin,152.41,71.85,6.00),v60,z5,tPen\WObj:=wPaper;
    MoveL Offs(pOrigin,156.07,69.81,6.00),vTravel,z5,tPen\WObj:=wPaper;
    MoveL Offs(pOrigin,156.07,69.81,0.00),v60,z0,tPen\WObj:=wPaper;
    MoveL Offs(pOrigin,154.80,69.81,0.00),v40,z0,tPen\WObj:=wPaper;
    MoveL Offs(pOrigin,153.31,69.32,0.00),v40,z0,tPen\WObj:=wPaper;
    MoveL Offs(pOrigin,152.60,68.11,0.00),v40,z0,tPen\WObj:=wPaper;
    MoveL Offs(pOrigin,152.89,67.90,0.00),v40,z0,tPen\WObj:=wPaper;
    MoveL Offs(pOrigin,155.01,68.47,0.00),v40,z0,tPen\WObj:=wPaper;
    MoveL Offs(pOrigin,156.07,69.39,0.00),v40,fine,tPen\WObj:=wPaper;
    MoveL Offs(pOrigin,156.07,69.39,6.00),v60,z5,tPen\WObj:=wPaper;
    MoveL Offs(pOrigin,163.69,68.54,6.00),vTravel,z5,tPen\WObj:=wPaper;
    MoveL Offs(pOrigin,163.69,68.54,0.00),v60,z0,tPen\WObj:=wPaper;
    MoveL Offs(pOrigin,163.69,70.24,0.00),v40,fine,tPen\WObj:=wPaper;
    MoveL Offs(pOrigin,163.69,70.24,6.00),v60,z5,tPen\WObj:=wPaper;
    MoveL Offs(pOrigin,148.55,59.28,6.00),vTravel,z5,tPen\WObj:=wPaper;
    MoveL Offs(pOrigin,148.55,59.28,0.00),v60,z0,tPen\WObj:=wPaper;
    MoveL Offs(pOrigin,142.24,65.59,0.00),v40,z0,tPen\WObj:=wPaper;
    MoveL Offs(pOrigin,142.90,64.93,0.00),v40,z0,tPen\WObj:=wPaper;
    MoveL Offs(pOrigin,143.54,65.56,0.00),v40,z0,tPen\WObj:=wPaper;
    MoveL Offs(pOrigin,142.90,64.93,0.00),v40,fine,tPen\WObj:=wPaper;
    MoveL Offs(pOrigin,142.90,64.93,6.00),v60,z5,tPen\WObj:=wPaper;
    MoveL Offs(pOrigin,144.18,64.29,6.00),vTravel,z5,tPen\WObj:=wPaper;
    MoveL Offs(pOrigin,144.18,64.29,0.00),v60,z0,tPen\WObj:=wPaper;
    MoveL Offs(pOrigin,140.99,60.67,0.00),v40,z0,tPen\WObj:=wPaper;
    MoveL Offs(pOrigin,140.99,60.67,0.00),v40,z0,tPen\WObj:=wPaper;
    MoveL Offs(pOrigin,140.85,59.61,0.00),v40,z0,tPen\WObj:=wPaper;
    MoveL Offs(pOrigin,139.43,56.85,0.00),v40,z0,tPen\WObj:=wPaper;
    MoveL Offs(pOrigin,138.58,54.30,0.00),v40,z0,tPen\WObj:=wPaper;
    MoveL Offs(pOrigin,137.38,52.81,0.00),v40,z0,tPen\WObj:=wPaper;
    MoveL Offs(pOrigin,137.38,52.81,0.00),v40,z0,tPen\WObj:=wPaper;
    MoveL Offs(pOrigin,137.16,53.88,0.00),v40,z0,tPen\WObj:=wPaper;
    MoveL Offs(pOrigin,138.15,57.28,0.00),v40,z0,tPen\WObj:=wPaper;
    MoveL Offs(pOrigin,139.50,59.61,0.00),v40,z0,tPen\WObj:=wPaper;
    MoveL Offs(pOrigin,140.35,60.53,0.00),v40,z0,tPen\WObj:=wPaper;
    MoveL Offs(pOrigin,140.99,60.67,0.00),v40,fine,tPen\WObj:=wPaper;
    MoveL Offs(pOrigin,140.99,60.67,6.00),v60,z5,tPen\WObj:=wPaper;
    MoveL Offs(pOrigin,140.78,59.35,6.00),vTravel,z5,tPen\WObj:=wPaper;
    MoveL Offs(pOrigin,140.78,59.35,0.00),v60,z0,tPen\WObj:=wPaper;
    MoveL Offs(pOrigin,146.94,59.35,0.00),v40,z0,tPen\WObj:=wPaper;
    MoveL Offs(pOrigin,147.79,59.40,0.00),v40,z0,tPen\WObj:=wPaper;
    MoveL Offs(pOrigin,148.00,59.83,0.00),v40,z0,tPen\WObj:=wPaper;
    MoveL Offs(pOrigin,147.79,59.40,0.00),v40,z0,tPen\WObj:=wPaper;
    MoveL Offs(pOrigin,147.81,58.53,0.00),v40,z0,tPen\WObj:=wPaper;
    MoveL Offs(pOrigin,141.35,64.99,0.00),v40,fine,tPen\WObj:=wPaper;
    MoveL Offs(pOrigin,141.35,64.99,6.00),v60,z5,tPen\WObj:=wPaper;
    MoveL Offs(pOrigin,144.69,65.99,6.00),vTravel,z5,tPen\WObj:=wPaper;
    MoveL Offs(pOrigin,144.69,65.99,0.00),v60,z0,tPen\WObj:=wPaper;
    MoveL Offs(pOrigin,144.69,62.80,0.00),v40,fine,tPen\WObj:=wPaper;
    MoveL Offs(pOrigin,144.69,62.80,6.00),v60,z5,tPen\WObj:=wPaper;
    MoveL Offs(pOrigin,146.80,62.16,6.00),vTravel,z5,tPen\WObj:=wPaper;
    MoveL Offs(pOrigin,146.80,62.16,0.00),v60,z0,tPen\WObj:=wPaper;
    MoveL Offs(pOrigin,146.80,60.25,0.00),v40,fine,tPen\WObj:=wPaper;
    MoveL Offs(pOrigin,146.80,60.25,6.00),v60,z5,tPen\WObj:=wPaper;
    MoveL Offs(pOrigin,144.69,58.76,6.00),vTravel,z5,tPen\WObj:=wPaper;
    MoveL Offs(pOrigin,144.69,58.76,0.00),v60,z0,tPen\WObj:=wPaper;
    MoveL Offs(pOrigin,144.69,57.06,0.00),v40,z0,tPen\WObj:=wPaper;
    MoveL Offs(pOrigin,143.63,56.85,0.00),v40,z0,tPen\WObj:=wPaper;
    MoveL Offs(pOrigin,143.63,54.51,0.00),v40,fine,tPen\WObj:=wPaper;
    MoveL Offs(pOrigin,143.63,54.51,6.00),v60,z5,tPen\WObj:=wPaper;
  ENDPROC

  PROC DrawPart292()
    MoveL Offs(pOrigin,140.56,52.17,6.00),vTravel,z5,tPen\WObj:=wPaper;
    MoveL Offs(pOrigin,140.56,52.17,0.00),v60,z0,tPen\WObj:=wPaper;
    MoveL Offs(pOrigin,139.29,52.17,0.00),v40,fine,tPen\WObj:=wPaper;
    MoveL Offs(pOrigin,139.29,52.17,6.00),v60,z5,tPen\WObj:=wPaper;
    MoveL Offs(pOrigin,137.29,52.81,6.00),vTravel,z5,tPen\WObj:=wPaper;
    MoveL Offs(pOrigin,137.29,52.81,0.00),v60,z0,tPen\WObj:=wPaper;
    MoveL Offs(pOrigin,137.29,48.56,0.00),v40,z0,tPen\WObj:=wPaper;
    MoveL Offs(pOrigin,136.74,48.79,0.00),v40,z0,tPen\WObj:=wPaper;
    MoveL Offs(pOrigin,138.44,48.79,0.00),v40,fine,tPen\WObj:=wPaper;
    MoveL Offs(pOrigin,138.44,48.79,6.00),v60,z5,tPen\WObj:=wPaper;
    MoveL Offs(pOrigin,135.71,48.23,6.00),vTravel,z5,tPen\WObj:=wPaper;
    MoveL Offs(pOrigin,135.71,48.23,0.00),v60,z0,tPen\WObj:=wPaper;
    MoveL Offs(pOrigin,149.08,34.86,0.00),v40,z0,tPen\WObj:=wPaper;
    MoveL Offs(pOrigin,148.82,35.61,0.00),v40,z0,tPen\WObj:=wPaper;
    MoveL Offs(pOrigin,153.33,40.12,0.00),v40,z0,tPen\WObj:=wPaper;
    MoveL Offs(pOrigin,153.13,39.21,0.00),v40,z0,tPen\WObj:=wPaper;
    MoveL Offs(pOrigin,153.13,37.09,0.00),v40,fine,tPen\WObj:=wPaper;
    MoveL Offs(pOrigin,153.13,37.09,6.00),v60,z5,tPen\WObj:=wPaper;
    MoveL Offs(pOrigin,152.08,38.79,6.00),vTravel,z5,tPen\WObj:=wPaper;
    MoveL Offs(pOrigin,152.08,38.79,0.00),v60,z0,tPen\WObj:=wPaper;
    MoveL Offs(pOrigin,152.08,39.85,0.00),v40,z0,tPen\WObj:=wPaper;
    MoveL Offs(pOrigin,151.02,40.28,0.00),v40,z0,tPen\WObj:=wPaper;
    MoveL Offs(pOrigin,151.02,38.79,0.00),v40,fine,tPen\WObj:=wPaper;
    MoveL Offs(pOrigin,151.02,38.79,6.00),v60,z5,tPen\WObj:=wPaper;
    MoveL Offs(pOrigin,148.84,41.61,6.00),vTravel,z5,tPen\WObj:=wPaper;
    MoveL Offs(pOrigin,148.84,41.61,0.00),v60,z0,tPen\WObj:=wPaper;
    MoveL Offs(pOrigin,142.98,35.75,0.00),v40,z0,tPen\WObj:=wPaper;
    MoveL Offs(pOrigin,142.94,35.03,0.00),v40,z0,tPen\WObj:=wPaper;
    MoveL Offs(pOrigin,139.03,38.94,0.00),v40,z0,tPen\WObj:=wPaper;
    MoveL Offs(pOrigin,139.24,37.98,0.00),v40,z0,tPen\WObj:=wPaper;
    MoveL Offs(pOrigin,137.74,36.48,0.00),v40,z0,tPen\WObj:=wPaper;
    MoveL Offs(pOrigin,137.84,35.64,0.00),v40,z0,tPen\WObj:=wPaper;
    MoveL Offs(pOrigin,132.58,40.90,0.00),v40,z0,tPen\WObj:=wPaper;
    MoveL Offs(pOrigin,131.61,40.80,0.00),v40,z0,tPen\WObj:=wPaper;
    MoveL Offs(pOrigin,128.15,37.35,0.00),v40,z0,tPen\WObj:=wPaper;
    MoveL Offs(pOrigin,128.10,36.42,0.00),v40,z0,tPen\WObj:=wPaper;
    MoveL Offs(pOrigin,118.64,45.89,0.00),v40,fine,tPen\WObj:=wPaper;
    MoveL Offs(pOrigin,118.64,45.89,6.00),v60,z5,tPen\WObj:=wPaper;
    MoveL Offs(pOrigin,119.52,47.74,6.00),vTravel,z5,tPen\WObj:=wPaper;
    MoveL Offs(pOrigin,119.52,47.74,0.00),v60,z0,tPen\WObj:=wPaper;
    MoveL Offs(pOrigin,121.01,47.74,0.00),v40,fine,tPen\WObj:=wPaper;
    MoveL Offs(pOrigin,121.01,47.74,6.00),v60,z5,tPen\WObj:=wPaper;
    MoveL Offs(pOrigin,121.65,50.90,6.00),vTravel,z5,tPen\WObj:=wPaper;
    MoveL Offs(pOrigin,121.65,50.90,0.00),v60,z0,tPen\WObj:=wPaper;
    MoveL Offs(pOrigin,119.74,50.90,0.00),v40,z0,tPen\WObj:=wPaper;
    MoveL Offs(pOrigin,119.74,51.96,0.00),v40,z0,tPen\WObj:=wPaper;
    MoveL Offs(pOrigin,121.86,51.96,0.00),v40,z0,tPen\WObj:=wPaper;
    MoveL Offs(pOrigin,121.45,52.39,0.00),v40,z0,tPen\WObj:=wPaper;
    MoveL Offs(pOrigin,121.45,54.30,0.00),v40,z0,tPen\WObj:=wPaper;
    MoveL Offs(pOrigin,122.07,54.30,0.00),v40,z0,tPen\WObj:=wPaper;
    MoveL Offs(pOrigin,122.29,54.72,0.00),v40,z0,tPen\WObj:=wPaper;
    MoveL Offs(pOrigin,122.07,54.30,0.00),v40,z0,tPen\WObj:=wPaper;
    MoveL Offs(pOrigin,122.50,54.07,0.00),v40,z0,tPen\WObj:=wPaper;
    MoveL Offs(pOrigin,120.16,54.07,0.00),v40,fine,tPen\WObj:=wPaper;
    MoveL Offs(pOrigin,120.16,54.07,6.00),v60,z5,tPen\WObj:=wPaper;
    MoveL Offs(pOrigin,120.59,56.18,6.00),vTravel,z5,tPen\WObj:=wPaper;
    MoveL Offs(pOrigin,120.59,56.18,0.00),v60,z0,tPen\WObj:=wPaper;
    MoveL Offs(pOrigin,122.08,56.18,0.00),v40,z0,tPen\WObj:=wPaper;
    MoveL Offs(pOrigin,122.29,57.24,0.00),v40,z0,tPen\WObj:=wPaper;
    MoveL Offs(pOrigin,121.01,57.24,0.00),v40,z0,tPen\WObj:=wPaper;
    MoveL Offs(pOrigin,120.10,57.87,0.00),v40,z0,tPen\WObj:=wPaper;
    MoveL Offs(pOrigin,125.66,52.31,0.00),v40,fine,tPen\WObj:=wPaper;
    MoveL Offs(pOrigin,125.66,52.31,6.00),v60,z5,tPen\WObj:=wPaper;
    MoveL Offs(pOrigin,125.80,53.66,6.00),vTravel,z5,tPen\WObj:=wPaper;
    MoveL Offs(pOrigin,125.80,53.66,0.00),v60,z0,tPen\WObj:=wPaper;
    MoveL Offs(pOrigin,120.54,58.92,0.00),v40,z0,tPen\WObj:=wPaper;
    MoveL Offs(pOrigin,121.65,59.35,0.00),v40,z0,tPen\WObj:=wPaper;
    MoveL Offs(pOrigin,123.14,59.35,0.00),v40,z0,tPen\WObj:=wPaper;
    MoveL Offs(pOrigin,123.35,59.61,0.00),v40,z0,tPen\WObj:=wPaper;
    MoveL Offs(pOrigin,123.56,60.04,0.00),v40,z0,tPen\WObj:=wPaper;
    MoveL Offs(pOrigin,123.35,59.61,0.00),v40,z0,tPen\WObj:=wPaper;
    MoveL Offs(pOrigin,123.78,60.25,0.00),v40,z0,tPen\WObj:=wPaper;
    MoveL Offs(pOrigin,125.90,62.38,0.00),v40,z0,tPen\WObj:=wPaper;
    MoveL Offs(pOrigin,123.78,60.25,0.00),v40,z0,tPen\WObj:=wPaper;
    MoveL Offs(pOrigin,123.99,60.41,0.00),v40,z0,tPen\WObj:=wPaper;
    MoveL Offs(pOrigin,122.29,60.41,0.00),v40,z0,tPen\WObj:=wPaper;
    MoveL Offs(pOrigin,122.07,60.25,0.00),v40,z0,tPen\WObj:=wPaper;
    MoveL Offs(pOrigin,122.71,61.10,0.00),v40,z0,tPen\WObj:=wPaper;
    MoveL Offs(pOrigin,122.07,60.25,0.00),v40,z0,tPen\WObj:=wPaper;
    MoveL Offs(pOrigin,121.93,61.00,0.00),v40,z0,tPen\WObj:=wPaper;
    MoveL Offs(pOrigin,125.54,64.60,0.00),v40,fine,tPen\WObj:=wPaper;
    MoveL Offs(pOrigin,125.54,64.60,6.00),v60,z5,tPen\WObj:=wPaper;
    MoveL Offs(pOrigin,125.05,61.46,6.00),vTravel,z5,tPen\WObj:=wPaper;
    MoveL Offs(pOrigin,125.05,61.46,0.00),v60,z0,tPen\WObj:=wPaper;
    MoveL Offs(pOrigin,123.14,61.46,0.00),v40,z0,tPen\WObj:=wPaper;
    MoveL Offs(pOrigin,122.18,61.76,0.00),v40,z0,tPen\WObj:=wPaper;
    MoveL Offs(pOrigin,126.99,56.95,0.00),v40,z0,tPen\WObj:=wPaper;
    MoveL Offs(pOrigin,126.54,55.90,0.00),v40,z0,tPen\WObj:=wPaper;
    MoveL Offs(pOrigin,121.59,60.86,0.00),v40,z0,tPen\WObj:=wPaper;
    MoveL Offs(pOrigin,120.84,60.11,0.00),v40,z0,tPen\WObj:=wPaper;
    MoveL Offs(pOrigin,126.25,54.70,0.00),v40,fine,tPen\WObj:=wPaper;
    MoveL Offs(pOrigin,126.25,54.70,6.00),v60,z5,tPen\WObj:=wPaper;
    MoveL Offs(pOrigin,125.66,55.77,6.00),vTravel,z5,tPen\WObj:=wPaper;
    MoveL Offs(pOrigin,125.66,55.77,0.00),v60,z0,tPen\WObj:=wPaper;
    MoveL Offs(pOrigin,124.31,54.41,0.00),v40,fine,tPen\WObj:=wPaper;
    MoveL Offs(pOrigin,124.31,54.41,6.00),v60,z5,tPen\WObj:=wPaper;
    MoveL Offs(pOrigin,125.66,50.81,6.00),vTravel,z5,tPen\WObj:=wPaper;
    MoveL Offs(pOrigin,125.66,50.81,0.00),v60,z0,tPen\WObj:=wPaper;
    MoveL Offs(pOrigin,119.65,56.82,0.00),v40,fine,tPen\WObj:=wPaper;
    MoveL Offs(pOrigin,119.65,56.82,6.00),v60,z5,tPen\WObj:=wPaper;
    MoveL Offs(pOrigin,121.65,41.97,6.00),vTravel,z5,tPen\WObj:=wPaper;
    MoveL Offs(pOrigin,121.65,41.97,0.00),v60,z0,tPen\WObj:=wPaper;
    MoveL Offs(pOrigin,122.29,40.49,0.00),v40,fine,tPen\WObj:=wPaper;
    MoveL Offs(pOrigin,122.29,40.49,6.00),v60,z5,tPen\WObj:=wPaper;
    MoveL Offs(pOrigin,123.57,40.70,6.00),vTravel,z5,tPen\WObj:=wPaper;
    MoveL Offs(pOrigin,123.57,40.70,0.00),v60,z0,tPen\WObj:=wPaper;
    MoveL Offs(pOrigin,123.57,39.42,0.00),v40,fine,tPen\WObj:=wPaper;
    MoveL Offs(pOrigin,123.57,39.42,6.00),v60,z5,tPen\WObj:=wPaper;
    MoveL Offs(pOrigin,124.62,40.49,6.00),vTravel,z5,tPen\WObj:=wPaper;
    MoveL Offs(pOrigin,124.62,40.49,0.00),v60,z0,tPen\WObj:=wPaper;
    MoveL Offs(pOrigin,123.35,41.76,0.00),v40,z0,tPen\WObj:=wPaper;
    MoveL Offs(pOrigin,124.62,40.49,0.00),v40,fine,tPen\WObj:=wPaper;
    MoveL Offs(pOrigin,124.62,40.49,6.00),v60,z5,tPen\WObj:=wPaper;
    MoveL Offs(pOrigin,125.69,41.40,6.00),vTravel,z5,tPen\WObj:=wPaper;
    MoveL Offs(pOrigin,125.69,41.40,0.00),v60,z0,tPen\WObj:=wPaper;
    MoveL Offs(pOrigin,129.72,41.40,0.00),v40,fine,tPen\WObj:=wPaper;
    MoveL Offs(pOrigin,129.72,41.40,6.00),v60,z5,tPen\WObj:=wPaper;
    MoveL Offs(pOrigin,133.12,39.85,6.00),vTravel,z5,tPen\WObj:=wPaper;
    MoveL Offs(pOrigin,133.12,39.85,0.00),v60,z0,tPen\WObj:=wPaper;
    MoveL Offs(pOrigin,133.55,39.64,0.00),v40,z0,tPen\WObj:=wPaper;
  ENDPROC

  PROC DrawPart293()
    MoveL Offs(pOrigin,133.12,39.85,0.00),v40,z0,tPen\WObj:=wPaper;
    MoveL Offs(pOrigin,133.07,39.21,0.00),v40,z0,tPen\WObj:=wPaper;
    MoveL Offs(pOrigin,133.07,37.51,0.00),v40,fine,tPen\WObj:=wPaper;
    MoveL Offs(pOrigin,133.07,37.51,6.00),v60,z5,tPen\WObj:=wPaper;
    MoveL Offs(pOrigin,137.22,42.24,6.00),vTravel,z5,tPen\WObj:=wPaper;
    MoveL Offs(pOrigin,137.22,42.24,0.00),v60,z0,tPen\WObj:=wPaper;
    MoveL Offs(pOrigin,144.43,35.02,0.00),v40,fine,tPen\WObj:=wPaper;
    MoveL Offs(pOrigin,144.43,35.02,6.00),v60,z5,tPen\WObj:=wPaper;
    MoveL Offs(pOrigin,149.36,42.05,6.00),vTravel,z5,tPen\WObj:=wPaper;
    MoveL Offs(pOrigin,149.36,42.05,0.00),v60,z0,tPen\WObj:=wPaper;
    MoveL Offs(pOrigin,156.42,34.99,0.00),v40,fine,tPen\WObj:=wPaper;
    MoveL Offs(pOrigin,156.42,34.99,6.00),v60,z5,tPen\WObj:=wPaper;
    MoveL Offs(pOrigin,157.66,35.49,6.00),vTravel,z5,tPen\WObj:=wPaper;
    MoveL Offs(pOrigin,157.66,35.49,0.00),v60,z0,tPen\WObj:=wPaper;
    MoveL Offs(pOrigin,159.01,36.84,0.00),v40,fine,tPen\WObj:=wPaper;
    MoveL Offs(pOrigin,159.01,36.84,6.00),v60,z5,tPen\WObj:=wPaper;
    MoveL Offs(pOrigin,161.55,33.41,6.00),vTravel,z5,tPen\WObj:=wPaper;
    MoveL Offs(pOrigin,161.55,33.41,0.00),v60,z0,tPen\WObj:=wPaper;
    MoveL Offs(pOrigin,162.75,34.61,0.00),v40,fine,tPen\WObj:=wPaper;
    MoveL Offs(pOrigin,162.75,34.61,6.00),v60,z5,tPen\WObj:=wPaper;
    MoveL Offs(pOrigin,161.81,42.40,6.00),vTravel,z5,tPen\WObj:=wPaper;
    MoveL Offs(pOrigin,161.81,42.40,0.00),v60,z0,tPen\WObj:=wPaper;
    MoveL Offs(pOrigin,161.81,46.86,0.00),v40,z0,tPen\WObj:=wPaper;
    MoveL Offs(pOrigin,162.45,49.62,0.00),v40,fine,tPen\WObj:=wPaper;
    MoveL Offs(pOrigin,162.45,49.62,6.00),v60,z5,tPen\WObj:=wPaper;
    MoveL Offs(pOrigin,145.45,44.95,6.00),vTravel,z5,tPen\WObj:=wPaper;
    MoveL Offs(pOrigin,145.45,44.95,0.00),v60,z0,tPen\WObj:=wPaper;
    MoveL Offs(pOrigin,144.60,45.38,0.00),v40,z0,tPen\WObj:=wPaper;
    MoveL Offs(pOrigin,144.60,46.65,0.00),v40,fine,tPen\WObj:=wPaper;
    MoveL Offs(pOrigin,144.60,46.65,6.00),v60,z5,tPen\WObj:=wPaper;
    MoveL Offs(pOrigin,138.01,42.83,6.00),vTravel,z5,tPen\WObj:=wPaper;
    MoveL Offs(pOrigin,138.01,42.83,0.00),v60,z0,tPen\WObj:=wPaper;
    MoveL Offs(pOrigin,137.80,43.25,0.00),v40,z0,tPen\WObj:=wPaper;
    MoveL Offs(pOrigin,138.01,42.83,0.00),v40,fine,tPen\WObj:=wPaper;
    MoveL Offs(pOrigin,138.01,42.83,6.00),v60,z5,tPen\WObj:=wPaper;
    MoveL Offs(pOrigin,125.90,41.55,6.00),vTravel,z5,tPen\WObj:=wPaper;
    MoveL Offs(pOrigin,125.90,41.55,0.00),v60,z0,tPen\WObj:=wPaper;
    MoveL Offs(pOrigin,126.11,41.12,0.00),v40,z0,tPen\WObj:=wPaper;
    MoveL Offs(pOrigin,125.90,41.55,0.00),v40,fine,tPen\WObj:=wPaper;
    MoveL Offs(pOrigin,125.90,41.55,6.00),v60,z5,tPen\WObj:=wPaper;
    MoveL Offs(pOrigin,109.54,29.23,6.00),vTravel,z5,tPen\WObj:=wPaper;
    MoveL Offs(pOrigin,109.54,29.23,0.00),v60,z0,tPen\WObj:=wPaper;
    MoveL Offs(pOrigin,109.32,29.44,0.00),v40,z0,tPen\WObj:=wPaper;
    MoveL Offs(pOrigin,107.41,29.23,0.00),v40,fine,tPen\WObj:=wPaper;
    MoveL Offs(pOrigin,107.41,29.23,6.00),v60,z5,tPen\WObj:=wPaper;
    MoveL Offs(pOrigin,103.87,30.98,6.00),vTravel,z5,tPen\WObj:=wPaper;
    MoveL Offs(pOrigin,103.87,30.98,0.00),v60,z0,tPen\WObj:=wPaper;
    MoveL Offs(pOrigin,98.16,25.27,0.00),v40,z0,tPen\WObj:=wPaper;
    MoveL Offs(pOrigin,98.03,24.68,0.00),v40,z0,tPen\WObj:=wPaper;
    MoveL Offs(pOrigin,88.41,34.30,0.00),v40,fine,tPen\WObj:=wPaper;
    MoveL Offs(pOrigin,88.41,34.30,6.00),v60,z5,tPen\WObj:=wPaper;
    MoveL Offs(pOrigin,87.66,33.05,6.00),vTravel,z5,tPen\WObj:=wPaper;
    MoveL Offs(pOrigin,87.66,33.05,0.00),v60,z0,tPen\WObj:=wPaper;
    MoveL Offs(pOrigin,87.66,31.99,0.00),v40,fine,tPen\WObj:=wPaper;
    MoveL Offs(pOrigin,87.66,31.99,6.00),v60,z5,tPen\WObj:=wPaper;
    MoveL Offs(pOrigin,85.52,31.90,6.00),vTravel,z5,tPen\WObj:=wPaper;
    MoveL Offs(pOrigin,85.52,31.90,0.00),v60,z0,tPen\WObj:=wPaper;
    MoveL Offs(pOrigin,90.41,31.90,0.00),v40,fine,tPen\WObj:=wPaper;
    MoveL Offs(pOrigin,90.41,31.90,6.00),v60,z5,tPen\WObj:=wPaper;
    MoveL Offs(pOrigin,98.06,41.34,6.00),vTravel,z5,tPen\WObj:=wPaper;
    MoveL Offs(pOrigin,98.06,41.34,0.00),v60,z0,tPen\WObj:=wPaper;
    MoveL Offs(pOrigin,98.49,41.12,0.00),v40,z0,tPen\WObj:=wPaper;
    MoveL Offs(pOrigin,98.06,41.34,0.00),v40,fine,tPen\WObj:=wPaper;
    MoveL Offs(pOrigin,98.06,41.34,6.00),v60,z5,tPen\WObj:=wPaper;
    MoveL Offs(pOrigin,99.34,42.40,6.00),vTravel,z5,tPen\WObj:=wPaper;
    MoveL Offs(pOrigin,99.34,42.40,0.00),v60,z0,tPen\WObj:=wPaper;
    MoveL Offs(pOrigin,99.76,42.19,0.00),v40,z0,tPen\WObj:=wPaper;
    MoveL Offs(pOrigin,99.34,42.40,0.00),v40,fine,tPen\WObj:=wPaper;
    MoveL Offs(pOrigin,99.34,42.40,6.00),v60,z5,tPen\WObj:=wPaper;
    MoveL Offs(pOrigin,95.97,45.49,6.00),vTravel,z5,tPen\WObj:=wPaper;
    MoveL Offs(pOrigin,95.97,45.49,0.00),v60,z0,tPen\WObj:=wPaper;
    MoveL Offs(pOrigin,94.47,43.99,0.00),v40,fine,tPen\WObj:=wPaper;
    MoveL Offs(pOrigin,94.47,43.99,6.00),v60,z5,tPen\WObj:=wPaper;
    MoveL Offs(pOrigin,94.96,48.66,6.00),vTravel,z5,tPen\WObj:=wPaper;
    MoveL Offs(pOrigin,94.96,48.66,0.00),v60,z0,tPen\WObj:=wPaper;
    MoveL Offs(pOrigin,91.35,52.26,0.00),v40,fine,tPen\WObj:=wPaper;
    MoveL Offs(pOrigin,91.35,52.26,6.00),v60,z5,tPen\WObj:=wPaper;
    MoveL Offs(pOrigin,92.11,54.07,6.00),vTravel,z5,tPen\WObj:=wPaper;
    MoveL Offs(pOrigin,92.11,54.07,0.00),v60,z0,tPen\WObj:=wPaper;
    MoveL Offs(pOrigin,94.88,54.07,0.00),v40,fine,tPen\WObj:=wPaper;
    MoveL Offs(pOrigin,94.88,54.07,6.00),v60,z5,tPen\WObj:=wPaper;
    MoveL Offs(pOrigin,94.66,55.58,6.00),vTravel,z5,tPen\WObj:=wPaper;
    MoveL Offs(pOrigin,94.66,55.58,0.00),v60,z0,tPen\WObj:=wPaper;
    MoveL Offs(pOrigin,94.45,56.21,0.00),v40,z0,tPen\WObj:=wPaper;
    MoveL Offs(pOrigin,96.36,61.53,0.00),v40,z0,tPen\WObj:=wPaper;
    MoveL Offs(pOrigin,96.36,62.38,0.00),v40,fine,tPen\WObj:=wPaper;
    MoveL Offs(pOrigin,96.36,62.38,6.00),v60,z5,tPen\WObj:=wPaper;
    MoveL Offs(pOrigin,94.88,60.89,6.00),vTravel,z5,tPen\WObj:=wPaper;
    MoveL Offs(pOrigin,94.88,60.89,0.00),v60,z0,tPen\WObj:=wPaper;
    MoveL Offs(pOrigin,95.09,61.31,0.00),v40,z0,tPen\WObj:=wPaper;
    MoveL Offs(pOrigin,94.88,60.89,0.00),v40,z0,tPen\WObj:=wPaper;
    MoveL Offs(pOrigin,94.17,61.39,0.00),v40,z0,tPen\WObj:=wPaper;
    MoveL Offs(pOrigin,97.63,57.94,0.00),v40,z0,tPen\WObj:=wPaper;
    MoveL Offs(pOrigin,96.57,58.34,0.00),v40,z0,tPen\WObj:=wPaper;
    MoveL Offs(pOrigin,96.79,59.61,0.00),v40,z0,tPen\WObj:=wPaper;
    MoveL Offs(pOrigin,97.21,59.61,0.00),v40,fine,tPen\WObj:=wPaper;
    MoveL Offs(pOrigin,97.21,59.61,6.00),v60,z5,tPen\WObj:=wPaper;
    MoveL Offs(pOrigin,95.72,59.35,6.00),vTravel,z5,tPen\WObj:=wPaper;
    MoveL Offs(pOrigin,95.72,59.35,0.00),v60,z0,tPen\WObj:=wPaper;
    MoveL Offs(pOrigin,94.45,59.35,0.00),v40,z0,tPen\WObj:=wPaper;
    MoveL Offs(pOrigin,94.45,60.04,0.00),v40,z0,tPen\WObj:=wPaper;
    MoveL Offs(pOrigin,94.66,60.46,0.00),v40,z0,tPen\WObj:=wPaper;
    MoveL Offs(pOrigin,94.45,60.04,0.00),v40,z0,tPen\WObj:=wPaper;
    MoveL Offs(pOrigin,93.72,60.35,0.00),v40,z0,tPen\WObj:=wPaper;
    MoveL Offs(pOrigin,97.18,56.89,0.00),v40,fine,tPen\WObj:=wPaper;
    MoveL Offs(pOrigin,97.18,56.89,6.00),v60,z5,tPen\WObj:=wPaper;
    MoveL Offs(pOrigin,95.51,58.30,6.00),vTravel,z5,tPen\WObj:=wPaper;
    MoveL Offs(pOrigin,95.51,58.30,0.00),v60,z0,tPen\WObj:=wPaper;
    MoveL Offs(pOrigin,93.81,58.30,0.00),v40,fine,tPen\WObj:=wPaper;
    MoveL Offs(pOrigin,93.81,58.30,6.00),v60,z5,tPen\WObj:=wPaper;
    MoveL Offs(pOrigin,97.64,64.93,6.00),vTravel,z5,tPen\WObj:=wPaper;
    MoveL Offs(pOrigin,97.64,64.93,0.00),v60,z0,tPen\WObj:=wPaper;
    MoveL Offs(pOrigin,97.85,65.35,0.00),v40,z0,tPen\WObj:=wPaper;
    MoveL Offs(pOrigin,97.64,64.93,0.00),v40,fine,tPen\WObj:=wPaper;
    MoveL Offs(pOrigin,97.64,64.93,6.00),v60,z5,tPen\WObj:=wPaper;
    MoveL Offs(pOrigin,95.19,69.33,6.00),vTravel,z5,tPen\WObj:=wPaper;
    MoveL Offs(pOrigin,95.19,69.33,0.00),v60,z0,tPen\WObj:=wPaper;
    MoveL Offs(pOrigin,93.39,71.13,0.00),v40,z0,tPen\WObj:=wPaper;
    MoveL Offs(pOrigin,93.84,72.18,0.00),v40,z0,tPen\WObj:=wPaper;
    MoveL Offs(pOrigin,95.64,70.38,0.00),v40,z0,tPen\WObj:=wPaper;
  ENDPROC

  PROC DrawPart294()
    MoveL Offs(pOrigin,95.51,71.30,0.00),v40,z0,tPen\WObj:=wPaper;
    MoveL Offs(pOrigin,96.36,72.36,0.00),v40,z0,tPen\WObj:=wPaper;
    MoveL Offs(pOrigin,95.51,71.30,0.00),v40,z0,tPen\WObj:=wPaper;
    MoveL Offs(pOrigin,96.39,71.12,0.00),v40,z0,tPen\WObj:=wPaper;
    MoveL Offs(pOrigin,94.58,72.93,0.00),v40,z0,tPen\WObj:=wPaper;
    MoveL Offs(pOrigin,94.41,72.30,0.00),v40,z0,tPen\WObj:=wPaper;
    MoveL Offs(pOrigin,101.02,78.91,0.00),v40,fine,tPen\WObj:=wPaper;
    MoveL Offs(pOrigin,101.02,78.91,6.00),v60,z5,tPen\WObj:=wPaper;
    MoveL Offs(pOrigin,99.34,77.04,6.00),vTravel,z5,tPen\WObj:=wPaper;
    MoveL Offs(pOrigin,99.34,77.04,0.00),v60,z0,tPen\WObj:=wPaper;
    MoveL Offs(pOrigin,99.76,77.46,0.00),v40,z0,tPen\WObj:=wPaper;
    MoveL Offs(pOrigin,99.34,77.04,0.00),v40,fine,tPen\WObj:=wPaper;
    MoveL Offs(pOrigin,99.34,77.04,6.00),v60,z5,tPen\WObj:=wPaper;
    MoveL Offs(pOrigin,98.28,75.97,6.00),vTravel,z5,tPen\WObj:=wPaper;
    MoveL Offs(pOrigin,98.28,75.97,0.00),v60,z0,tPen\WObj:=wPaper;
    MoveL Offs(pOrigin,99.12,76.82,0.00),v40,z0,tPen\WObj:=wPaper;
    MoveL Offs(pOrigin,98.28,75.97,0.00),v40,z0,tPen\WObj:=wPaper;
    MoveL Offs(pOrigin,97.85,75.19,0.00),v40,z0,tPen\WObj:=wPaper;
    MoveL Offs(pOrigin,98.91,75.19,0.00),v40,z0,tPen\WObj:=wPaper;
    MoveL Offs(pOrigin,98.28,74.49,0.00),v40,z0,tPen\WObj:=wPaper;
    MoveL Offs(pOrigin,99.12,75.34,0.00),v40,z0,tPen\WObj:=wPaper;
    MoveL Offs(pOrigin,98.28,74.49,0.00),v40,z0,tPen\WObj:=wPaper;
    MoveL Offs(pOrigin,97.85,74.14,0.00),v40,z0,tPen\WObj:=wPaper;
    MoveL Offs(pOrigin,96.79,74.14,0.00),v40,z0,tPen\WObj:=wPaper;
    MoveL Offs(pOrigin,96.57,74.49,0.00),v40,z0,tPen\WObj:=wPaper;
    MoveL Offs(pOrigin,97.43,75.34,0.00),v40,z0,tPen\WObj:=wPaper;
    MoveL Offs(pOrigin,96.57,74.49,0.00),v40,z0,tPen\WObj:=wPaper;
    MoveL Offs(pOrigin,95.78,74.72,0.00),v40,z0,tPen\WObj:=wPaper;
    MoveL Offs(pOrigin,97.73,72.77,0.00),v40,z0,tPen\WObj:=wPaper;
    MoveL Offs(pOrigin,96.79,73.00,0.00),v40,z0,tPen\WObj:=wPaper;
    MoveL Offs(pOrigin,97.64,73.85,0.00),v40,z0,tPen\WObj:=wPaper;
    MoveL Offs(pOrigin,96.79,73.00,0.00),v40,z0,tPen\WObj:=wPaper;
    MoveL Offs(pOrigin,97.13,71.87,0.00),v40,z0,tPen\WObj:=wPaper;
    MoveL Offs(pOrigin,95.18,73.82,0.00),v40,fine,tPen\WObj:=wPaper;
    MoveL Offs(pOrigin,95.18,73.82,6.00),v60,z5,tPen\WObj:=wPaper;
    MoveL Offs(pOrigin,94.66,71.94,6.00),vTravel,z5,tPen\WObj:=wPaper;
    MoveL Offs(pOrigin,94.66,71.94,0.00),v60,z0,tPen\WObj:=wPaper;
    MoveL Offs(pOrigin,94.88,72.36,0.00),v40,z0,tPen\WObj:=wPaper;
    MoveL Offs(pOrigin,94.66,71.94,0.00),v40,fine,tPen\WObj:=wPaper;
    MoveL Offs(pOrigin,94.66,71.94,6.00),v60,z5,tPen\WObj:=wPaper;
    MoveL Offs(pOrigin,92.79,73.23,6.00),vTravel,z5,tPen\WObj:=wPaper;
    MoveL Offs(pOrigin,92.79,73.23,0.00),v60,z0,tPen\WObj:=wPaper;
    MoveL Offs(pOrigin,90.23,75.79,0.00),v40,z0,tPen\WObj:=wPaper;
    MoveL Offs(pOrigin,89.63,74.89,0.00),v40,z0,tPen\WObj:=wPaper;
    MoveL Offs(pOrigin,92.34,72.18,0.00),v40,fine,tPen\WObj:=wPaper;
    MoveL Offs(pOrigin,92.34,72.18,6.00),v60,z5,tPen\WObj:=wPaper;
    MoveL Offs(pOrigin,92.11,74.14,6.00),vTravel,z5,tPen\WObj:=wPaper;
    MoveL Offs(pOrigin,92.11,74.14,0.00),v60,z0,tPen\WObj:=wPaper;
    MoveL Offs(pOrigin,90.62,74.14,0.00),v40,fine,tPen\WObj:=wPaper;
    MoveL Offs(pOrigin,90.62,74.14,6.00),v60,z5,tPen\WObj:=wPaper;
    MoveL Offs(pOrigin,92.96,76.19,6.00),vTravel,z5,tPen\WObj:=wPaper;
    MoveL Offs(pOrigin,92.96,76.19,0.00),v60,z0,tPen\WObj:=wPaper;
    MoveL Offs(pOrigin,93.18,76.61,0.00),v40,z0,tPen\WObj:=wPaper;
    MoveL Offs(pOrigin,92.96,76.19,0.00),v40,fine,tPen\WObj:=wPaper;
    MoveL Offs(pOrigin,92.96,76.19,6.00),v60,z5,tPen\WObj:=wPaper;
    MoveL Offs(pOrigin,94.27,76.22,6.00),vTravel,z5,tPen\WObj:=wPaper;
    MoveL Offs(pOrigin,94.27,76.22,0.00),v60,z0,tPen\WObj:=wPaper;
    MoveL Offs(pOrigin,91.87,78.63,0.00),v40,z0,tPen\WObj:=wPaper;
    MoveL Offs(pOrigin,92.75,78.36,0.00),v40,z0,tPen\WObj:=wPaper;
    MoveL Offs(pOrigin,94.45,78.36,0.00),v40,z0,tPen\WObj:=wPaper;
    MoveL Offs(pOrigin,94.45,78.53,0.00),v40,z0,tPen\WObj:=wPaper;
    MoveL Offs(pOrigin,94.66,78.95,0.00),v40,z0,tPen\WObj:=wPaper;
    MoveL Offs(pOrigin,94.45,78.53,0.00),v40,fine,tPen\WObj:=wPaper;
    MoveL Offs(pOrigin,94.45,78.53,6.00),v60,z5,tPen\WObj:=wPaper;
    MoveL Offs(pOrigin,93.06,80.42,6.00),vTravel,z5,tPen\WObj:=wPaper;
    MoveL Offs(pOrigin,93.06,80.42,0.00),v60,z0,tPen\WObj:=wPaper;
    MoveL Offs(pOrigin,99.37,74.11,0.00),v40,z0,tPen\WObj:=wPaper;
    MoveL Offs(pOrigin,98.48,73.51,0.00),v40,z0,tPen\WObj:=wPaper;
    MoveL Offs(pOrigin,96.52,75.47,0.00),v40,fine,tPen\WObj:=wPaper;
    MoveL Offs(pOrigin,96.52,75.47,6.00),v60,z5,tPen\WObj:=wPaper;
    MoveL Offs(pOrigin,123.61,84.22,6.00),vTravel,z5,tPen\WObj:=wPaper;
    MoveL Offs(pOrigin,123.61,84.22,0.00),v60,z0,tPen\WObj:=wPaper;
    MoveL Offs(pOrigin,126.77,81.07,0.00),v40,fine,tPen\WObj:=wPaper;
    MoveL Offs(pOrigin,126.77,81.07,6.00),v60,z5,tPen\WObj:=wPaper;
    MoveL Offs(pOrigin,130.71,89.19,6.00),vTravel,z5,tPen\WObj:=wPaper;
    MoveL Offs(pOrigin,130.71,89.19,0.00),v60,z0,tPen\WObj:=wPaper;
    MoveL Offs(pOrigin,132.81,91.29,0.00),v40,fine,tPen\WObj:=wPaper;
    MoveL Offs(pOrigin,132.81,91.29,6.00),v60,z5,tPen\WObj:=wPaper;
    MoveL Offs(pOrigin,144.20,92.22,6.00),vTravel,z5,tPen\WObj:=wPaper;
    MoveL Offs(pOrigin,144.20,92.22,0.00),v60,z0,tPen\WObj:=wPaper;
    MoveL Offs(pOrigin,145.10,93.13,0.00),v40,fine,tPen\WObj:=wPaper;
    MoveL Offs(pOrigin,145.10,93.13,6.00),v60,z5,tPen\WObj:=wPaper;
    MoveL Offs(pOrigin,139.50,59.40,6.00),vTravel,z5,tPen\WObj:=wPaper;
    MoveL Offs(pOrigin,139.50,59.40,0.00),v60,z0,tPen\WObj:=wPaper;
    MoveL Offs(pOrigin,140.14,60.04,0.00),v40,z0,tPen\WObj:=wPaper;
    MoveL Offs(pOrigin,139.50,59.40,0.00),v40,z0,tPen\WObj:=wPaper;
    MoveL Offs(pOrigin,139.50,59.35,0.00),v40,z0,tPen\WObj:=wPaper;
    MoveL Offs(pOrigin,138.01,59.35,0.00),v40,z0,tPen\WObj:=wPaper;
    MoveL Offs(pOrigin,137.80,59.40,0.00),v40,z0,tPen\WObj:=wPaper;
    MoveL Offs(pOrigin,138.01,59.83,0.00),v40,z0,tPen\WObj:=wPaper;
    MoveL Offs(pOrigin,137.80,59.40,0.00),v40,fine,tPen\WObj:=wPaper;
    MoveL Offs(pOrigin,137.80,59.40,6.00),v60,z5,tPen\WObj:=wPaper;
    MoveL Offs(pOrigin,142.26,58.12,6.00),vTravel,z5,tPen\WObj:=wPaper;
    MoveL Offs(pOrigin,142.26,58.12,0.00),v60,z0,tPen\WObj:=wPaper;
    MoveL Offs(pOrigin,142.48,58.55,0.00),v40,z0,tPen\WObj:=wPaper;
    MoveL Offs(pOrigin,142.26,58.12,0.00),v40,fine,tPen\WObj:=wPaper;
    MoveL Offs(pOrigin,142.26,58.12,6.00),v60,z5,tPen\WObj:=wPaper;
    MoveL Offs(pOrigin,151.49,26.33,6.00),vTravel,z5,tPen\WObj:=wPaper;
    MoveL Offs(pOrigin,151.49,26.33,0.00),v60,z0,tPen\WObj:=wPaper;
    MoveL Offs(pOrigin,145.48,20.32,0.00),v40,fine,tPen\WObj:=wPaper;
    MoveL Offs(pOrigin,145.48,20.32,6.00),v60,z5,tPen\WObj:=wPaper;
    MoveL Offs(pOrigin,173.84,117.62,6.00),vTravel,z5,tPen\WObj:=wPaper;
    MoveL Offs(pOrigin,173.84,117.62,0.00),v60,z0,tPen\WObj:=wPaper;
    MoveL Offs(pOrigin,172.04,119.43,0.00),v40,z0,tPen\WObj:=wPaper;
    MoveL Offs(pOrigin,172.48,120.47,0.00),v40,z0,tPen\WObj:=wPaper;
    MoveL Offs(pOrigin,174.44,118.52,0.00),v40,fine,tPen\WObj:=wPaper;
    MoveL Offs(pOrigin,174.44,118.52,6.00),v60,z5,tPen\WObj:=wPaper;
    MoveL Offs(pOrigin,170.99,120.48,6.00),vTravel,z5,tPen\WObj:=wPaper;
    MoveL Offs(pOrigin,170.99,120.48,0.00),v60,z0,tPen\WObj:=wPaper;
    MoveL Offs(pOrigin,170.08,121.38,0.00),v40,z0,tPen\WObj:=wPaper;
    MoveL Offs(pOrigin,169.34,120.63,0.00),v40,z0,tPen\WObj:=wPaper;
    MoveL Offs(pOrigin,170.39,119.58,0.00),v40,fine,tPen\WObj:=wPaper;
    MoveL Offs(pOrigin,170.39,119.58,6.00),v60,z5,tPen\WObj:=wPaper;
    MoveL Offs(pOrigin,176.26,124.85,6.00),vTravel,z5,tPen\WObj:=wPaper;
    MoveL Offs(pOrigin,176.26,124.85,0.00),v60,z0,tPen\WObj:=wPaper;
    MoveL Offs(pOrigin,176.48,125.28,0.00),v40,z0,tPen\WObj:=wPaper;
    MoveL Offs(pOrigin,176.26,124.85,0.00),v40,z0,tPen\WObj:=wPaper;
    MoveL Offs(pOrigin,177.32,124.85,0.00),v40,z0,tPen\WObj:=wPaper;
    MoveL Offs(pOrigin,177.54,125.28,0.00),v40,z0,tPen\WObj:=wPaper;
    MoveL Offs(pOrigin,177.32,124.85,0.00),v40,fine,tPen\WObj:=wPaper;
  ENDPROC

  PROC DrawPart295()
    MoveL Offs(pOrigin,177.32,124.85,6.00),v60,z5,tPen\WObj:=wPaper;
    MoveL Offs(pOrigin,130.60,148.91,6.00),vTravel,z5,tPen\WObj:=wPaper;
    MoveL Offs(pOrigin,130.60,148.91,0.00),v60,z0,tPen\WObj:=wPaper;
    MoveL Offs(pOrigin,128.35,151.17,0.00),v40,fine,tPen\WObj:=wPaper;
    MoveL Offs(pOrigin,128.35,151.17,6.00),v60,z5,tPen\WObj:=wPaper;
    MoveL Offs(pOrigin,128.79,153.71,6.00),vTravel,z5,tPen\WObj:=wPaper;
    MoveL Offs(pOrigin,128.79,153.71,0.00),v60,z0,tPen\WObj:=wPaper;
    MoveL Offs(pOrigin,131.49,151.01,0.00),v40,fine,tPen\WObj:=wPaper;
    MoveL Offs(pOrigin,131.49,151.01,6.00),v60,z5,tPen\WObj:=wPaper;
  ENDPROC

ENDMODULE
